// TIA Portal V18 export
DATA_BLOCK "04_SPEED"   // DB6, F_DB
{ S7_Optimized_Access := 'TRUE'; DB_Accessible_From_OPC_UA := 'FALSE' }
// stored: DBAccessibleFromOPCUA false
   VAR
      AlwaysFALSE : Bool;
      AlwaysTRUE : Bool := TRUE;
      "!!ITERATOR_STRINGS$$" : Bool;
      "!!04_SPEED.{db_element:ENC1/2}$$" : Bool;
      "!!04_SPEED.{db_element:ENC2/2}$$" : Bool;
      "!!04_SPEED.{db_element:ENC}$$" : Bool;
   END_VAR
BEGIN
END_DATA_BLOCK
